FUNCTION F_ComputeRawVarint64Size : UDINT
VAR_INPUT
    nValue : ULINT;
END_VAR
VAR
    i       : UDINT;
    nMask   : ULINT;
END_VAR


FOR i := 1 TO 9 DO    
    nMask := SHL(16#FFFFFFFFFFFFFFFF, 7 * i);
    IF (nValue AND nMask) = 0 THEN
        F_ComputeRawVarint64Size := i;
        RETURN;
    END_IF
END_FOR

F_ComputeRawVarint64Size := 10;

END_FUNCTION

(* stored: Version 1.1.0.1
   POU F_ComputeRawVarint64Size: Id {53f9253e-b577-4ce6-bc41-aefb89dd7733}, SpecialFunc None *)
